// TIA Portal project "S7-1500 İlk Proje" (V18)

(* hardware
DEVICE "S7-1500/ET200MP station_1"  S7-1500 station
   slot 0: "Rail_0"  Rack  6ES7 590-1***0-0AA0
   slot 1: "PLC_1"  CPU 1512C-1 PN  6ES7 512-1CK01-0AB0  V2.8
      slot 3: "CPU display_1"  6ES7591-1AA00-0AA0
      slot 32768: "PROFINET interface_1"  X1
         slot 32769: "Port_1"  X1 P1
         slot 32770: "Port_2"  X1 P2
      slot 34817: "Virtual CP interface port_1"  Virtual CP interface port  Virtual CP interface port
DEVICE "HMI_1"  KTP700 Basic PN
   slot 0: "HMI_1"  KTP700 Basic PN  6AV2 123-2GB03-0AX0  14.0.1.0
   slot 1: "HMI_RT_1"  KTP700 Basic PN  6AV2 123-2GB03-0AX0  14.0.1.0
   slot 5: "HMI_1.IE_CP_1"  PROFINET Interface  14.0.1.0
      slot 1: "PROFINET Interface_1"  PROFINET Interface
         slot 1: "Port_1"  Port
*)

// ===== PLC "PLC_1"  CPU 1512C-1 PN =====

VAR_GLOBAL   // PLC tag table "Default tag table"
   "Motor" AT %Q0.0 : Bool;
   "Stop" AT %I0.0 : Bool;
   "Start" AT %I0.1 : Bool;
END_VAR

ORGANIZATION_BLOCK "Main"   // OB1, LAD, ProgramCycle
TITLE = "Main Program Sweep (Cycle)"
{ S7_Optimized_Access := 'TRUE' }
VERSION : 0.1
   VAR_INPUT
      Initial_Call : Bool;   // Initial call of this OB
      Remanence : Bool;   // =True, if remanent data are available
   END_VAR
BEGIN

REGION Network 1
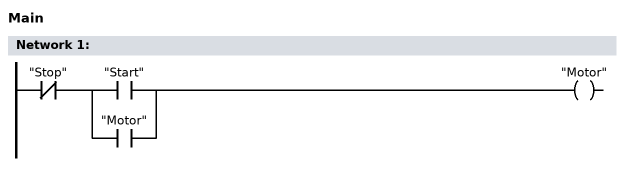
   RUNG wire#powerrail
      I_Contact( "Stop" )
      wire#w1
      Contact( "Start" )
      wire#w2
      Coil( "Motor" )
   END_RUNG
   RUNG wire#w1
      Contact( "Motor" )
   END_RUNG wire#w2
   // the same network as SCL:
   "Motor" := NOT "Stop" AND ("Start" OR "Motor");
END_REGION
END_ORGANIZATION_BLOCK

(* ===== HMI "HMI_RT_1" =====
system functions are stored by id; their names below are inferred from use
connection "Connection_1": ETHERNET, SMART_S7_1500_OMS

HMI tags "Default tag table"
   "Tag_ScreenNumber" : UInt, internal
   "Stop" : Bool AT %I0.0, 100 ms
   "Start" : Bool AT %I0.1, 100 ms
   "Motor" : Bool AT %Q0.0, 100 ms

graphic list "Motor": 0 'Graphic_1'; 1 'Graphic_2'

Template "Template_1" 800x480
   Button "Exit" at 714,429 size 71x50; TextOff 'Exit'; PictureOff "ExitRuntime_KTP700_Basic_PN_TR"; PictureOn "ExitRuntime_KTP700_Basic_PN_TR"
      on Release: StopRuntime(0)
   Button "Language" at 614,429 size 71x50; TextOff 'Language'; PictureOff "ToggleLanguage_KTP700_Basic_PN_TR"; PictureOn "ToggleLanguage_KTP700_Basic_PN_TR"
      on Release: function_fb9197e8(-1)
   Button "Log on" at 514,429 size 71x50; TextOff 'Log on'; PictureOff "Login_KTP700_Basic_PN_TR"; PictureOn "Login_KTP700_Basic_PN_TR"
      on Release: function_a2a04561()
   Button "Alarms" at 114,429 size 71x50; TextOff 'Alarms'; PictureOff "AlarmDisplay_KTP700_Basic_PN_TR"; PictureOn "AlarmDisplay_KTP700_Basic_PN_TR"
      on Release: function_ef3f5d25("Alarm window_Unacknowledged", -1)
   Button "Start screen" at 14,429 size 71x50; TextOff 'Start screen'; PictureOff "NavigateHome_KTP700_Basic_PN_TR"; PictureOn "NavigateHome_KTP700_Basic_PN_TR"
      on Release: ActivateScreen("Root screen", 0)
   SymbolicIOField "Symbolic_IO_Field_Screen" at 93,9 size 600x33; TextOff '0'; TextOn '1'; TextList "TextList_ScreenNames"
      ProcessValue <- "Tag_ScreenNumber"
      on Change: ActivateScreenByNumber("Tag_ScreenNumber", 0)
   DateTimeField "HmiScreenItemData" at 695,25 size 105x25
   DateTimeField "HmiScreenItemData_1" at 695,0 size 105x25
   GraphicView "Logo" at 0,0 size 91x51; Picture "Logo of HMI_1"

screen "Root screen" 800x480, template "Template_1"
   on GenerateScreen: SetTag("Tag_ScreenNumber", 1)
   TextField "HmiScreenItemData" at 68,75 size 644x25; Text 'S7-1500 PLC Eğitim Seti İlk WinCC Projesi'
   Button "Button_1" at 209,130 size 141x79; TextOff 'Start'
      on Click: SetBit("Motor"); SetBit("Start")
   Button "Button_2" at 209,221 size 141x79; TextOff 'Stop'
      on Click: ResetBit("Motor"); SetBit("Stop")
   GraphicIOField "Graphic I/O field_1" at 370,130 size 203x169; PictureList "Motor"
      ProcessValue <- "Motor"
*)